(* IEC 61131-3 sources: IRIS-Project/LASAL CONTROL SOFTWARE/LasalProject_2025_09_12/Class/Attuatore, 1 file *)

(* ---- Attuatore.st ---- *)
(*!
<Class
	Name               = "Attuatore"
	Revision           = "0.0"
	RealtimeTask       = "false"
	CyclicTask         = "true"
	DefCyclictime      = "100 ms"
	BackgroundTask     = "false"
	Sigmatek           = "false"
	OSInterface        = "false"
	HighPriority       = "false"
	Automatic          = "false"
	UpdateMode         = "Prescan"
	SharedCommandTable = "true"
	Objectsize         = "(676,120)">
	<Channels>
		<Server Name="ClassSvr" Visualized="false" Initialize="false" WriteProtected="true" Retentive="false"/>
		<Server Name="s_Solenoid_Command" Visualized="false" Initialize="false" WriteProtected="false" Retentive="false"/>
		<Server Name="s_Solenoid_Status" Visualized="false" Initialize="false" WriteProtected="false" Retentive="false"/>
		<Server Name="s_State" Visualized="false" Initialize="false" WriteProtected="false" Retentive="false"/>
		<Client Name="R_aus_1" Required="true" Internal="false"/>
		<Client Name="R_aus_2" Required="true" Internal="false"/>
		<Client Name="R_p" Required="true" Internal="false"/>
	</Channels>
</Class>
*)
Attuatore : CLASS
	TYPE
	  t_fsm_actuator :  //! <Type Public="true" Name="t_fsm_actuator"/>
	  (
	    idle,
	    Push,
	    Pull
	  )$UDINT;
	END_TYPE
  //Servers:
	ClassSvr 	: SvrChCmd_DINT;
	s_Solenoid_Command 	: SvrCh_DINT;
	s_State 	: SvrCh_DINT;
	s_Solenoid_Status 	: SvrCh_DINT;
  //Clients:
	R_p 	: CltCh_DINT;
	R_aus_1 	: CltCh_DINT;
	R_aus_2 	: CltCh_DINT;
  //Variables:
		fsm_step 	: t_fsm_actuator;
		Tempo 	: DINT;
		Status 	: BOOL;
		Command 	: DINT;
  //Functions:

	FUNCTION VIRTUAL GLOBAL Init;

	FUNCTION VIRTUAL GLOBAL CyWork
		VAR_INPUT
			EAX 	: UDINT;
		END_VAR
		VAR_OUTPUT
			state (EAX) 	: UDINT;
		END_VAR;

	FUNCTION GLOBAL SetSequenceState
		VAR_INPUT
			Param 	: t_fsm_actuator;
		END_VAR
		VAR_OUTPUT
			retcode 	: DINT;
		END_VAR;

	FUNCTION GLOBAL GetActuatorStatus
		VAR_OUTPUT
			ActuatorStatus 	: DINT;
		END_VAR;

	FUNCTION VIRTUAL GLOBAL s_Solenoid_Command::Read
		VAR_OUTPUT
			output (EAX) 	: DINT;
		END_VAR;

	FUNCTION VIRTUAL GLOBAL s_State::Read
		VAR_OUTPUT
			output (EAX) 	: DINT;
		END_VAR;
  //Tables:
	FUNCTION @STD
		VAR_OUTPUT
			ret_code	: CONFSTATES;
		END_VAR;
	FUNCTION GLOBAL TAB @CT_;
END_CLASS;

FUNCTION VIRTUAL GLOBAL Attuatore::CyWork
	VAR_INPUT
		EAX 	: UDINT;
	END_VAR
	VAR_OUTPUT
		state (EAX) 	: UDINT;
	END_VAR

 Command:=s_Solenoid_Command.Read();
 s_Solenoid_Status.Write(input:=Status);

 if Command=0 then
    fsm_step:=idle;
 elsif Command=1 then
    fsm_step:=Push;
 elsif Command=2 then
    fsm_step:=Pull;
 end_if;

case fsm_step of

  Idle://Idle
  Tempo:=0;
  //Status:=2; //Idle

  Push: //ESTRATTO
      Tempo:=Tempo+100;

      if Tempo=1000 then
         R_aus_1.Write(input:=1);
      end_if;

      if Tempo=1500 then
        R_aus_1.Write(input:=0);
        Status:=1; //pushed
        fsm_step:=Idle;
        Tempo:=0;
        Command:=3;
        s_Solenoid_Command.Write(input:=3);
      end_if;

  Pull: //RETRATTO
      Tempo:=Tempo+100;

      IF R_aus_1=0 & Tempo=1000 THEN
        R_p.Write(input:=1);
      END_IF;

      if R_aus_1=0 & Tempo=1500 then
         R_aus_2.Write(input:=1);
      end_if;

      if tempo=2500 then
        R_aus_2.Write(input:=0);
        R_p.Write(input:=0);
        Status:=0; //pulled
        Tempo:=0;
        fsm_step:=Idle;
        Command:=3;
        s_Solenoid_Command.Write(input:=3);
      end_if;

  end_case;

	state := READY;

END_FUNCTION

FUNCTION VIRTUAL GLOBAL Attuatore::Init
Tempo:=0;
Command:=3;
Status:=FALSE; // false->pulled || true->pushed

END_FUNCTION

FUNCTION GLOBAL Attuatore::SetSequenceState
	VAR_INPUT
		Param 	: t_fsm_actuator;
	END_VAR
	VAR_OUTPUT
		retcode 	: DINT;
	END_VAR

  fsm_step:=Param;
  if fsm_step=Push then
    s_Solenoid_Command.Write(input:=1);
  elsif fsm_step=Pull then
    s_Solenoid_Command.Write(input:=2);
  end_if;
  retcode:=TRUE;

END_FUNCTION

FUNCTION GLOBAL Attuatore::GetActuatorStatus
	VAR_OUTPUT
		ActuatorStatus 	: DINT;
	END_VAR
  ActuatorStatus:=Status;
END_FUNCTION

FUNCTION VIRTUAL GLOBAL Attuatore::s_Solenoid_Command::Read
	VAR_OUTPUT
		output (EAX) 	: DINT;
	END_VAR

	output := s_Solenoid_Command;

END_FUNCTION

FUNCTION VIRTUAL GLOBAL Attuatore::s_State::Read
	VAR_OUTPUT
		output (EAX) 	: DINT;
	END_VAR

	output := s_State;

END_FUNCTION
